{attribute addProperty BoxType "EL9930-0000-0017"}
{attribute addProperty Id "IO_InputsEMPTY_STRUCTURE000IO_OutputsEMPTY_STRUCTURE000WcStateAT %I*WcState_98A4DF7520.250InfoDataAT %I*InfoData_BC63D37F80100"}
{attribute addProperty CRC "4278957859"}
{attribute addProperty SizeInBites "82"}
{attribute addProperty SizeInBytes "10.25"}
TYPE EL9930_546406CD :
STRUCT
	{attribute addProperty Name "IO_Inputs"}
	IO_Inputs : EMPTY_STRUCTURE;
	{attribute addProperty Name "IO_Outputs"}
	IO_Outputs : EMPTY_STRUCTURE;
	{attribute addProperty Name "WcState"}
	WcState : WcState_98A4DF75;
	{attribute addProperty Name "InfoData"}
	InfoData : InfoData_BC63D37F;
END_STRUCT
END_TYPE

(* stored: Version 1.2.0.0, ProductVersion 3.1.4024.9
   DUT EL9930_546406CD: Id {804ffa15-77b1-4fff-90f2-ce4c3ca23925} *)
